Fanuc TP program (LS listing): M_EXE17.LS

/PROG  M_EXE17	  Macro
/ATTR
OWNER		= MNEDITOR;
COMMENT		= "Manual macro17";
PROG_SIZE	= 194;
CREATE		= DATE 22-03-26  TIME 13:11:58;
MODIFIED	= DATE 22-06-20  TIME 07:19:20;
FILE_NAME	= M_EXE12;
VERSION		= 0;
LINE_COUNT	= 1;
MEMORY_SIZE	= 570;
PROTECT		= READ_WRITE;
TCD:  STACK_SIZE	= 0,
      TASK_PRIORITY	= 50,
      TIME_SLICE	= 0,
      BUSY_LAMP_OFF	= 0,
      ABORT_REQUEST	= 0,
      PAUSE_REQUEST	= 0;
DEFAULT_GROUP	= 1,*,*,*,*;
CONTROL_CODE	= 00000000 00000000;
/APPL
/APPL
/MN
   1:  CALL ROUTER(7) ;
/POS
/END
